TYPE ST_GCSpinAxisMoveVelCtrl EXTENDS ST_ServiceCtrlBase:
STRUCT
	Param : ST_GCSpinAxisMoveVelParam;
END_STRUCT
END_TYPE

(* stored: Version 1.1.0.1, ProductVersion 3.1.4026.18
   DUT ST_GCSpinAxisMoveVelCtrl: Id {bca46df2-18c9-49a3-b76a-340b92902e6e} *)
